% RSLogix 500 project cascading_timers.RSS, saved by version 8.30.00.16 %
PROJECT "UNTITLED"    % processor: Bul.1763 MicroLogix 1100 Series B %

PROGRAM FILES
  LAD 2   7 rungs

DATA FILES
  O0 OUTPUT  4 elements
  I1 INPUT  6 elements
  S2 STATUS  66 elements
  B3 BINARY  1 elements
  T4 TIMER  2 elements
  C5 COUNTER  1 elements
  R6 CONTROL  1 elements
  N7 INTEGER  20 elements
  F8 FLOAT  1 elements
  N9 DELTATIMES  256 elements

LADDER 2
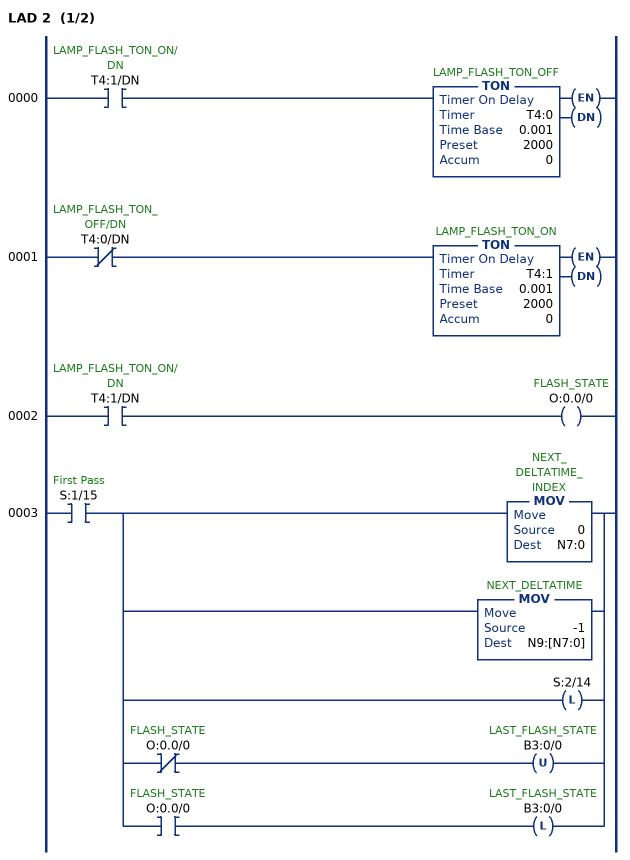
% Rung: 0 %
SOR XIC T4:1/DN TON T4:0 0.001 2000 0 EOR
%   T4:1  LAMP_FLASH_TON_ON %
%   T4:0  LAMP_FLASH_TON_OFF %
% Rung: 1 %
SOR XIO T4:0/DN TON T4:1 0.001 2000 0 EOR
%   T4:0  LAMP_FLASH_TON_OFF %
%   T4:1  LAMP_FLASH_TON_ON %
% Rung: 2 %
SOR XIC T4:1/DN OTE O:0.0/0 EOR
%   T4:1  LAMP_FLASH_TON_ON %
%   O:0.0/0  FLASH_STATE %
% Rung: 3 %
SOR XIC S:1/15 BST MOV 0 N7:0 NXB MOV -1 N9:[N7:0] NXB OTL S:2/14 NXB XIO O:0.0/0 OTU B3:0/0 NXB XIC O:0.0/0 OTL B3:0/0 BND EOR
%   S:1/15  "First Pass" %
%   N7:0  NEXT_DELTATIME_INDEX %
%   N9:[N7:0]  NEXT_DELTATIME %
%   O:0.0/0  FLASH_STATE %
%   B3:0/0  LAST_FLASH_STATE %

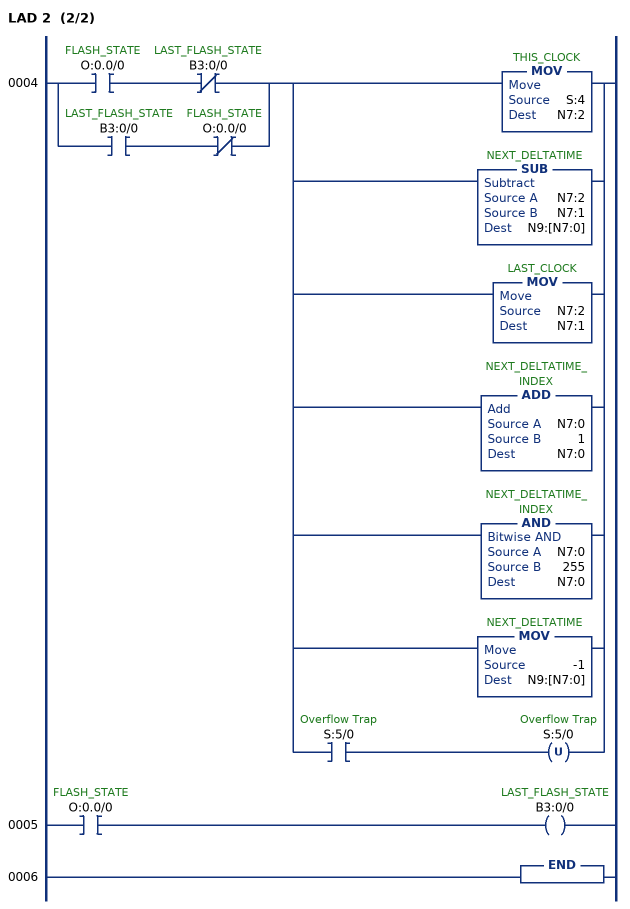
% Rung: 4 %
SOR BST XIC O:0.0/0 XIO B3:0/0 NXB XIC B3:0/0 XIO O:0.0/0 BND BST MOV S:4 N7:2 NXB SUB N7:2 N7:1 N9:[N7:0] NXB MOV N7:2 N7:1 NXB ADD N7:0 1 N7:0 NXB AND N7:0 255 N7:0 NXB MOV -1 N9:[N7:0] NXB XIC S:5/0 OTU S:5/0 BND EOR
%   O:0.0/0  FLASH_STATE %
%   B3:0/0  LAST_FLASH_STATE %
%   S:4  "Time Base" %
%   N7:2  THIS_CLOCK %
%   N7:1  LAST_CLOCK %
%   N9:[N7:0]  NEXT_DELTATIME %
%   N7:0  NEXT_DELTATIME_INDEX %
%   S:5/0  "Overflow Trap" %
% Rung: 5 %
SOR XIC O:0.0/0 OTE B3:0/0 EOR
%   O:0.0/0  FLASH_STATE %
%   B3:0/0  LAST_FLASH_STATE %
% Rung: 6 %
SOR END EOR

OTHER DOCUMENTED ADDRESSES
  I:0.0/[N7:1]  TANK_BY_INDEX_STATE
  RTC:0.SEC/1  LAMP_FLASH_RTC_BIT01

DATA TABLE (non-zero values as saved)
DATA T4
% .PRE .ACC %
% T4:0 % 2000 0
% T4:1 % 2000 0
